Yaskawa INFORM job: R2_O2(0,-90).JBI

/JOB
//NAME R2_O2(0,-90)
///FOLDERNAME X4
//POS
///NPOS 49,49,49,2,0,0
///TOOL 0
///POSTYPE PULSE
///PULSE
C00000=-165077,-11048,-3465,42103,97235,-25872
C00001=-162183,-9836,-336,42374,94865,-25532
C00002=-161029,-9262,990,42486,93918,-25400
C00003=-160152,-10314,166,42597,93469,-25188
C00004=-161029,-9262,990,42486,93918,-25400
C00005=-155810,-567,4500,35086,99149,-23871
C00006=-155808,-23,6235,34998,98496,-24080
C00007=-155810,-567,4500,35086,99149,-23871
C00008=-165621,-20133,-4325,46072,91900,-27108
C00009=-162746,-23856,-7550,46453,90473,-26404
C00010=-162169,-22096,-6308,46528,90273,-26221
C00011=-162746,-23856,-7550,46453,90473,-26404
C00012=-165621,-20133,-4325,46072,91900,-27108
C00013=-163520,-13167,830,46368,91107,-26476
C00014=-164758,-13802,-430,46230,92061,-26621
C00015=-167869,-15166,-3399,45891,94455,-26994
C00016=-151938,-52542,-29763,49238,79071,17279
C00017=-120607,-73680,-36955,53746,51644,75521
C00018=-120606,-71360,-32677,54675,50777,74846
C00019=-120606,-70405,-30939,55060,50434,74570
C00020=-122338,-70380,-30926,55241,51412,74153
C00021=-120609,-71426,-32794,54650,50801,74863
C00022=-120606,-70415,-30957,55056,50437,74573
C00023=-120606,-70429,-30984,55050,50442,74577
C00024=-120606,-70439,-31002,55046,50446,74580
C00025=-120606,-71394,-32740,54661,50790,74856
C00026=-120607,-73713,-37016,53732,51657,75530
C00027=-120607,-73914,-37421,53641,51745,75598
C00028=-120606,-71605,-33154,54565,50877,74925
C00029=-120606,-70654,-31420,54948,50533,74650
C00030=-122338,-70629,-31407,55132,51511,74233
C00031=-120609,-71671,-33271,54540,50901,74943
C00032=-120606,-70675,-31458,54939,50540,74656
C00033=-120606,-71625,-33192,54556,50885,74931
C00034=-120607,-73934,-37458,53633,51753,75603
C00035=-130128,-72407,-43401,39669,56587,31237
C00036=-120641,-15578,-8997,18341,54391,-34113
C00037=-120641,-14559,-5716,18683,52969,-34377
C00038=-120641,-14119,-4373,18828,52399,-34486
C00039=-120339,-16187,-6381,18643,52494,-34334
C00040=-121492,-13717,-4673,19132,52967,-34752
C00041=-120642,-10963,4465,37761,35155,-44390
C00042=-120643,-10962,4466,49416,32859,-47789
C00043=-120645,-10956,4470,62920,31465,-52022
C00044=-120646,-10953,4472,75290,33021,-52557
C00045=-120648,-10941,4482,87100,34672,-52796
C00046=-120649,-10930,4490,87100,34673,-52796
C00047=-120649,-10935,4486,87100,34673,-52796
C00048=-120649,-10949,4476,87101,34673,-52797
BC00000=393560,699530,1075175
BC00001=393560,699530,1075175
BC00002=393560,699530,1075175
BC00003=393560,699530,1075175
BC00004=393560,699530,1075175
BC00005=393560,699530,1075175
BC00006=393560,699530,1075175
BC00007=393560,699530,1075175
BC00008=393560,699530,1075175
BC00009=393560,699530,1075175
BC00010=393560,699530,1075175
BC00011=393560,699530,1075175
BC00012=393560,699530,1075175
BC00013=393560,699530,1075175
BC00014=393560,699530,1075175
BC00015=393560,699530,1075175
BC00016=347924,712047,1075175
BC00017=292398,738338,1075175
BC00018=298016,739023,1075175
BC00019=300264,739297,1075175
BC00020=300264,739297,1075175
BC00021=300264,739297,1075175
BC00022=300273,743906,1075175
BC00023=300287,750372,1075175
BC00024=300296,754980,1075175
BC00025=298049,754706,1075175
BC00026=292430,754020,1075175
BC00027=299634,726271,1075175
BC00028=305253,726957,1075175
BC00029=307500,727231,1075175
BC00030=307500,727231,1075175
BC00031=307500,727231,1075175
BC00032=307520,736683,1075175
BC00033=305273,736408,1075175
BC00034=299654,735723,1075175
BC00035=319371,709844,1075175
BC00036=328570,645961,1075175
BC00037=333053,650417,1075175
BC00038=334846,652200,1075175
BC00039=334846,652200,1075175
BC00040=334846,652200,1075175
BC00041=323843,632241,1026959
BC00042=317252,628473,987061
BC00043=311367,625699,941836
BC00044=304910,625774,898310
BC00045=301100,625849,851704
BC00046=301098,625880,830117
BC00047=298876,623747,828203
BC00048=293321,618417,823416
EC00000=0,-556475
EC00001=0,-556475
EC00002=0,-556475
EC00003=0,-556475
EC00004=0,-556475
EC00005=0,-556475
EC00006=0,-556475
EC00007=0,-556475
EC00008=0,-556475
EC00009=0,-556475
EC00010=0,-556475
EC00011=0,-556475
EC00012=0,-556475
EC00013=0,-556475
EC00014=0,-556475
EC00015=0,-556475
EC00016=0,-556475
EC00017=0,-556475
EC00018=0,-556475
EC00019=0,-556475
EC00020=0,-556475
EC00021=0,-556475
EC00022=0,-556475
EC00023=0,-556475
EC00024=0,-556475
EC00025=0,-556475
EC00026=0,-556475
EC00027=0,-556475
EC00028=0,-556475
EC00029=0,-556475
EC00030=0,-556475
EC00031=0,-556475
EC00032=0,-556475
EC00033=0,-556475
EC00034=0,-556475
EC00035=0,-556475
EC00036=0,-556475
EC00037=0,-556475
EC00038=0,-556475
EC00039=0,-556475
EC00040=0,-556475
EC00041=0,-556475
EC00042=0,-556475
EC00043=0,-556475
EC00044=0,-556475
EC00045=0,-556475
EC00046=0,-556475
EC00047=0,-556475
EC00048=0,-556475
///POSTYPE BASE
///RECTAN
///RCONF 0,0,0,0,0,0,0,0,0,0,0,0,0,0,0,0,0,0,0,0,0,0,0,0
P00006=0.222,-3.123,-1.508,0.0000,0.0000,0.0000
P00021=-0.225,-6.128,-0.405,0.0000,0.0000,0.0000
//INST
///DATE 2023/12/15 10:19
///ATTR SC,RW
///GROUP1 RB1,BS1
///GROUP2 ST1
NOP
'r2_O2(0,-90)
'Path S1191
SSFTOF
MOVJ C00000 BC00000 VJ=100.00  +MOVJ EC00000 VJ=100.00
MOVL C00001 BC00001 V=400.0  +MOVJ EC00001 VJ=100.00
SMOVL C00002 BC00002 V=60.0  +MOVJ EC00002
SREFP 3 C00003 BC00003  +REFP EC00003
CALL JOB:SEARCH-R1-S1
SET P021 P006
SSFTON P021
SMOVL C00004 BC00004 V=60.0  +MOVJ EC00004
SMOVL C00005 BC00005 V=60.0  +MOVJ EC00005
SREFP 3 C00006 BC00006  +REFP EC00006
CALL JOB:SEARCH-R1-S1
SET P021 P006
SSFTON P021
SMOVL C00007 BC00007 V=60.0  +MOVJ EC00007
SMOVL C00008 BC00008 V=100.0  +MOVJ EC00008
SMOVL C00009 BC00009 V=60.0  +MOVJ EC00009
SREFP 3 C00010 BC00010  +REFP EC00010
CALL JOB:SEARCH-R1-S1
SET P021 P006
SSFTON P021
SMOVL C00011 BC00011 V=60.0  +MOVJ EC00011
SMOVL C00012 BC00012 V=100.0  +MOVJ EC00012
SMOVL C00013 BC00013 V=100.0  +MOVJ EC00013
MOVL C00014 BC00014 V=400.0  +MOVJ EC00014 VJ=100.00
MOVL C00015 BC00015 V=1000.0  +MOVJ EC00015 VJ=100.00
'Path VIA1202
SSFTOF
MOVJ C00016 BC00016 VJ=100.00  +MOVJ EC00016 VJ=100.00
'Path W1192
SSFTOF
SSFTON P021
MOVJ C00017 BC00017 VJ=100.00  +MOVJ EC00017 VJ=100.00
SMOVL C00018 BC00018 V=400.0  +MOVJ EC00018
SMOVL C00019 BC00019 V=100.0 PL=0  +MOVJ EC00019
SREFP 1 C00020 BC00020  +REFP EC00020
SREFP 2 C00021 BC00021  +REFP EC00021
MACRO1 MJ#(0) ARGF0
ARCON
SMOVL C00022 BC00022 V=10.0  +MOVJ EC00022
SMOVL C00023 BC00023 V=10.0  +MOVJ EC00023
SMOVL C00024 BC00024 V=10.0  +MOVJ EC00024
ARCOF
SMOVL C00025 BC00025 V=400.0  +MOVJ EC00025
SMOVL C00026 BC00026 V=1000.0  +MOVJ EC00026
SSFTOF
'Path W1193
SSFTOF
SSFTON P021
MOVJ C00027 BC00027 VJ=100.00  +MOVJ EC00027 VJ=100.00
SMOVL C00028 BC00028 V=400.0  +MOVJ EC00028
SMOVL C00029 BC00029 V=100.0 PL=0  +MOVJ EC00029
SREFP 1 C00030 BC00030  +REFP EC00030
SREFP 2 C00031 BC00031  +REFP EC00031
MACRO1 MJ#(0) ARGF0
ARCON
SMOVL C00032 BC00032 V=10.0  +MOVJ EC00032
ARCOF
SMOVL C00033 BC00033 V=400.0  +MOVJ EC00033
SMOVL C00034 BC00034 V=1000.0  +MOVJ EC00034
SSFTOF
'Path VIA1203
SSFTOF
MOVJ C00035 BC00035 VJ=100.00  +MOVJ EC00035 VJ=100.00
'Path W1194
SSFTOF
SSFTON P021
MOVJ C00036 BC00036 VJ=100.00  +MOVJ EC00036 VJ=100.00
SMOVL C00037 BC00037 V=400.0  +MOVJ EC00037
SMOVL C00038 BC00038 V=100.0 PL=0  +MOVJ EC00038
SREFP 1 C00039 BC00039  +REFP EC00039
SREFP 2 C00040 BC00040  +REFP EC00040
MACRO1 MJ#(0) ARGF0
ARCON
SMOVL C00041 BC00041 V=10.0  +MOVJ EC00041
SMOVL C00042 BC00042 V=10.0  +MOVJ EC00042
SMOVL C00043 BC00043 V=10.0  +MOVJ EC00043
SMOVL C00044 BC00044 V=10.0  +MOVJ EC00044
SMOVL C00045 BC00045 V=10.0  +MOVJ EC00045
SMOVL C00046 BC00046 V=10.0  +MOVJ EC00046
ARCOF
SMOVL C00047 BC00047 V=400.0  +MOVJ EC00047
SMOVL C00048 BC00048 V=1000.0  +MOVJ EC00048
SSFTOF
END
